Universal Robots PolyScope program: Weight_Detection.urp

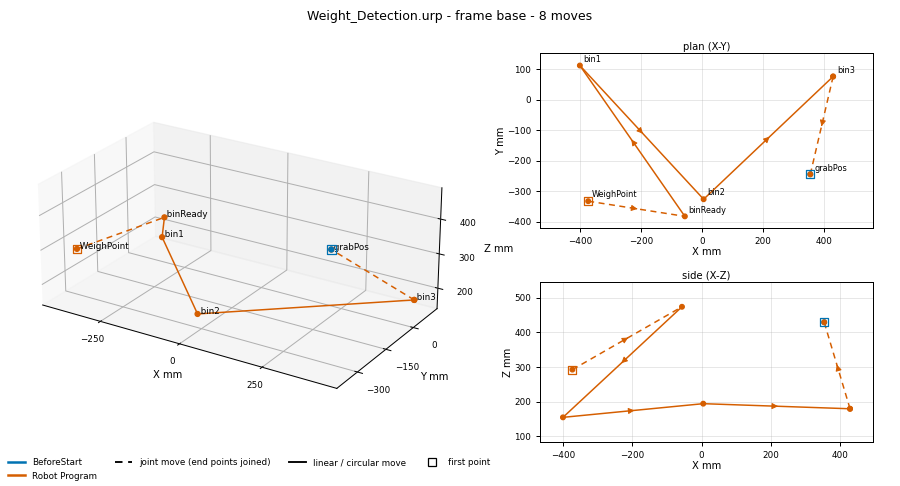
[picture p0: tool path of Weight_Detection.urp in frame base, 8 of 8 moves have a stored position in this frame; points joined in program order, loops and branches not executed]
Program Weight_Detection (installation=default directory=/programs/usbdisk_0/new folder_1 createdIn=5.8.0.10253 lastSavedIn=5.8.0.10253 robotSerialNumber=20205300708)
Calibrated DH parameters: a=[-0.000048, -0.164988, -0.190768, -0.000044, -0.000167, 0]; d=[0.151937, 265.766517, -282.786649, 17.1509, 0.085408, 0.091845]; alpha=[1.570475, 0.000674, 0.005589, 1.571818, -1.57228, 0]; deltaTheta=[0, 0.826521, -1.289102, 0.462588, 0, 0]
BeforeStart
  Set ExpressionOutput pin=ObjectWeight; expression=9999
  Set ExpressionOutput pin=SortingDone; expression=1
  Set ExpressionOutput pin=position; expression=0
  MoveJ speed 60 deg/s, acceleration 80 deg/s^2 (useActiveTCP=true) feature=Base
    Waypoint grabPos: TCP in base x=353.88 y=-243.828 z=429.304 mm, rx=1.7497 ry=1.6183 rz=-0.8122 rad; joints [-6.52, -115.268, -35, -114.309, -320.923, -904.659] deg
    Popup Warning (haltProgram=false message=Gripper will open and may drop something! inputType=Text)
    URCap Gripper Activate (Robotiq_Grippers, Robotiq Inc.) dataModel(ResetAndActivateKey=false)
    URCap Gripper (Robotiq_Grippers, Robotiq Inc.) dataModel(position=0.0, force=100.0, speed=100.0, positionInDouble=0.0, forceInDouble=100.0, speedInDouble=100.0, slaveIds=[9], blocking=true)
Robot Program (runOnlyOnce=false)
  Set ExpressionOutput pin=SortingDone; expression=0
  Popup Message (haltProgram=false message=Place object in gripper inputType=Text)
  ''
  URCap Gripper (Robotiq_Grippers, Robotiq Inc.) dataModel(position=100.0, force=100.0, speed=100.0, positionInDouble=100.0, forceInDouble=100.0, speedInDouble=100.0, slaveIds=[9], blocking=true)
  MoveJ speed 60 deg/s, acceleration 80 deg/s^2 (useActiveTCP=true) feature=Base
    Waypoint WeighPoint: TCP in base x=-373.129 y=-331.86 z=292.51 mm, rx=0.6282 ry=1.4698 rz=-0.5607 rad; joints [-133.92, -144.996, -35, -90, -179.679, -1077.385] deg
  Wait Sleep waitTime=1
  Set ExpressionOutput pin=position; expression=1
  Wait Condition expression=AnalysisDone≟1
  weight := (TWX_Weight/1000)
  SuppressedNode
    Popup Message (haltProgram=false inputType=Variable) variable=weight
  MoveJ speed 60 deg/s, acceleration 80 deg/s^2 (useActiveTCP=true) feature=Base
    Waypoint binReady: TCP in base x=-56.778 y=-381.525 z=473.901 mm, rx=0.5337 ry=2.208 rz=-0.2095 rad; joints [-88.472, -112.593, -35.02, -93.891, -226.105, -1039.522] deg
  Set ExpressionOutput pin=position; expression=0
  If weight<2
    MoveL speed 250 mm/s, acceleration 1200 mm/s^2 (useActiveTCP=true) feature=Base
      Waypoint bin1: TCP in base x=-400.367 y=112.137 z=154.671 mm, rx=1.8495 ry=1.8625 rz=-0.6144 rad; joints [-185.167, -127.171, -84.758, -61.609, -233.44, -6.419] deg
      Call SetDown
  ElseIf weight<4
    MoveL speed 250 mm/s, acceleration 1200 mm/s^2 (useActiveTCP=true) feature=Base
      Waypoint bin2: TCP in base x=4.658 y=-325.513 z=194.153 mm, rx=1.8713 ry=1.7472 rz=-0.706 rad; joints [-58.751, -100.398, -136.269, 2.31, -292.518, 118.194] deg
      Call SetDown
  ElseIf weight<6.6
    MoveL speed 250 mm/s, acceleration 1200 mm/s^2 (useActiveTCP=true) feature=Base
      Waypoint bin3: TCP in base x=428.509 y=76.173 z=179.45 mm, rx=1.9115 ry=1.8536 rz=-0.4988 rad; joints [33.54, -125.089, -73.87, -88.406, -297.655, 219.8] deg
      Call SetDown
  Else 
    Popup Warning (haltProgram=true message=Weight too heavy inputType=Text)
    MoveL speed 250 mm/s, acceleration 1200 mm/s^2 (useActiveTCP=true) feature=Base
      Waypoint bin3: TCP in base x=428.509 y=76.173 z=179.45 mm, rx=1.9115 ry=1.8536 rz=-0.4988 rad; joints [33.54, -125.089, -73.87, -88.406, -297.655, 219.8] deg
      Call SetDown
  Set ExpressionOutput pin=SortingDone; expression=1
  MoveJ speed 60 deg/s, acceleration 80 deg/s^2 (useActiveTCP=true) feature=Base
    Wait Sleep waitTime=1
    Waypoint grabPos: TCP in base x=353.88 y=-243.828 z=429.304 mm, rx=1.7497 ry=1.6183 rz=-0.8122 rad; joints [-6.52, -115.268, -35, -114.309, -320.923, -904.659] deg
SubProgram -> SetDown
SubProgram SetDown (keepSynchronizedWithDisk=false)
  MoveL speed 250 mm/s, acceleration 1200 mm/s^2 (useActiveTCP=true) feature=Base
    MoveDirectionNode (selectedDirection=ZMinus toolParams=0.05, 1.0)
      Until TOOL_CONTACT_DETECTION (allowActions=false retraction=0.007 decelerationAcceleration=3 decelerationAngularAcceleration=34.906585)
    URCap Gripper (Robotiq_Grippers, Robotiq Inc.) dataModel(position=0.0, force=100.0, speed=100.0, positionInDouble=0.0, forceInDouble=100.0, speedInDouble=100.0, slaveIds=[9], blocking=true)
    MoveDirectionNode expression=[0.0,1.0,1.0]
      Until DISTANCE (allowActions=false deceleration=3 distanceNodeType=STOP) Distance=0.05; motionParameters(blendRadius=0)
